FUNCTION_BLOCK RingTokenLogicConveyor7 (* Event-only Local Group Subscriber *)
  (* Standard: 61499-1; Classification: Communications; Description: Local Event Group Subscriber *)
  (* Version 0.1, 2002-05-02, JHC, Rockwell Automation, Optimized. *)
  (* Version 0.0, 2001-10-02, JHC, Rockwell Automation, Copied/modified from SUBSCRIBE *)
  (* Compiler header: package fb.rt.cs725; *)
  (* Compiler Java IBM VisualAge 3.0 *)
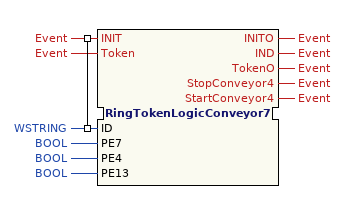
  EVENT_INPUT
    INIT WITH ID; (* Service Initialization *)
    Token;
  END_EVENT
  EVENT_OUTPUT
    INITO; (* Initialization Confirm *)
    IND; (* Service Indication *)
    TokenO;
    StopConveyor4;
    StartConveyor4;
  END_EVENT
  VAR_INPUT
    ID : WSTRING; (* Local Group Name-Default is FB Instance Name *)
    PE7 : BOOL;
    PE4 : BOOL;
    PE13 : BOOL;
  END_VAR
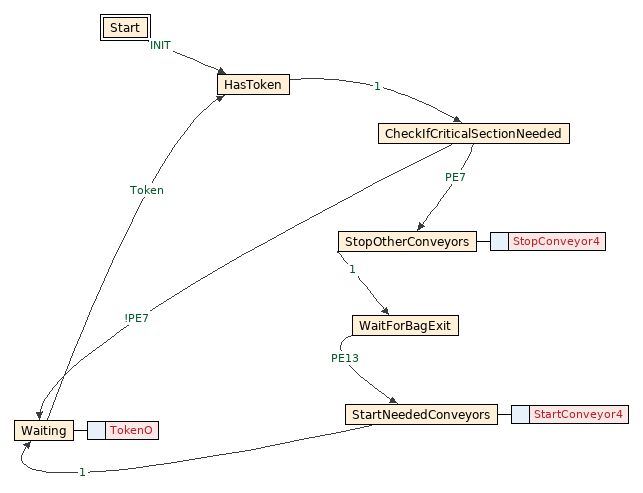
  EC_STATES
    Start; (* Has the token passed to it *)
    HasToken;
    Waiting : -> TokenO; (* When waiting for token *)
    CheckIfCriticalSectionNeeded;
    StopOtherConveyors : -> StopConveyor4;
    StartNeededConveyors : -> StartConveyor4;
    WaitForBagExit;
  END_STATES
  EC_TRANSITIONS
    Start TO HasToken := INIT;
    HasToken TO CheckIfCriticalSectionNeeded := 1;
    CheckIfCriticalSectionNeeded TO StopOtherConveyors := PE7;
    StartNeededConveyors TO Waiting := 1;
    Waiting TO HasToken := Token;
    CheckIfCriticalSectionNeeded TO Waiting := !PE7;
    StopOtherConveyors TO WaitForBagExit := 1;
    WaitForBagExit TO StartNeededConveyors := PE13;
  END_TRANSITIONS
  ALGORITHM NeedsCriticalSectionOrNot IN Java:

  END_ALGORITHM
END_FUNCTION_BLOCK
